// TIA Portal V18 export
TYPE "LGasp_typeCmdAttuatore"
// stored: IsFailsafeCompliant false
   STRUCT
      nome : WString[12];   // Nome assegnato all'attuatore = nome scritto su sequenza
      tipo : Int;   // 1=Ev, 2=Mot posizione, 3=HMC, 4=CNC (predisposizione), 5=Mot velocità, 6=Mot AAA
      savecorr : Bool;   // tasto salva correttore da HMI
      qset : LReal;   // Quota di destinazione nel caso di un asse
      corr : LReal;   // Correttore
      cmdhmi : "LGasp_typeCmdManAttuatore";   // Cmd start posizionamento
      cmdauto : "LGasp_typeCmdAutoAttuatore";   // Cmd start posizionamento
      sync { ExternalAccessible := 'False'; ExternalVisible := 'False'; ExternalWritable := 'False'} : "LGasp_typeSyncAttuatore";
   END_STRUCT;
END_TYPE
